(* IEC 61131-3 sources: repolevel_ST_code_completion/dataset/project_code/轴控/FB105_轴控制集/FC10_设备轴类, 3 files *)

(* ---- A01_通讯状态.st ---- *)
//从站通讯状态
pSlave := EtherCAT_Master_Leadshine.FirstSlave; //建立指针，指向主站后第一个从站
No_Slave:=0;
WHILE pSlave <> 0 DO
  No_Slave:=No_Slave+1;
  pSlave^(); //获取当前从站状态内容
IF pSlave^.wState <>ETC_SLAVE_STATE.ETC_SLAVE_OPERATIONAL THEN //
    ERROR[No_Slave]:=1;   //对应关系 ERROR[1]=1有错误   ERROR[1] 1号从站、ERROR[2] 2号从站,建立的数组元素个数等于从站个数
ELSE
    ERROR[No_Slave]:=0;
END_IF
pSlave := pSlave^.NextInstance; //指向下个从站，结尾为空，跳出循环
END_WHILE

//EtherCAT主站复位
EtherCAT_Master_Leadshine(
	xRestart:= bEtcReset,
	xStopBus:= ,
	xConfigFinished=> ,
	xDistributedClockInSync=> ,
	xError=> ,
	xSyncInWindow=> );

IF EtherCAT_Master_Leadshine.xConfigFinished AND EtherCAT_Master_Leadshine.xDistributedClockInSync THEN
	FB_AxisControl_AxisVirtual.ReStartSlaveEx:=TRUE;
	FB_AxisControl_调模A轴.ReStartSlaveEx:=TRUE;
	FB_AxisControl_调模B轴.ReStartSlaveEx:=TRUE;
	FB_AxisControl_送面料轴.ReStartSlaveEx:=TRUE;
	FB_AxisControl_取面料轴.ReStartSlaveEx:=TRUE;
	FB_AxisControl_横移A轴.ReStartSlaveEx:=TRUE;
	FB_AxisControl_升降A轴.ReStartSlaveEx:=TRUE;
	FB_AxisControl_横移B轴.ReStartSlaveEx:=TRUE;
	FB_AxisControl_升降B轴.ReStartSlaveEx:=TRUE;
	FB_AxisControl_出盒轴.ReStartSlaveEx:=TRUE;
	FB_AxisControl_铲灰板轴.ReStartSlaveEx:=TRUE;
	FB_AxisControl_包面纸轴.ReStartSlaveEx:=TRUE;
	FB_AxisControl_上包底轴.ReStartSlaveEx:=TRUE;
	FB_AxisControl_折边轴.ReStartSlaveEx:=TRUE;
	IF FB_AxisControl_AxisVirtual.ReStartSlaveDone AND FB_AxisControl_调模A轴.ReStartSlaveDone AND FB_AxisControl_调模B轴.ReStartSlaveDone AND
        FB_AxisControl_送面料轴.ReStartSlaveDone AND FB_AxisControl_取面料轴.ReStartSlaveDone AND FB_AxisControl_横移A轴.ReStartSlaveDone AND
		 FB_AxisControl_升降A轴.ReStartSlaveDone AND FB_AxisControl_横移B轴.ReStartSlaveDone AND FB_AxisControl_升降B轴.ReStartSlaveDone AND
		  FB_AxisControl_出盒轴.ReStartSlaveDone AND FB_AxisControl_铲灰板轴.ReStartSlaveDone AND FB_AxisControl_包面纸轴.ReStartSlaveDone AND
		   FB_AxisControl_上包底轴.ReStartSlaveDone AND FB_AxisControl_折边轴.ReStartSlaveDone THEN
	      bEtcReset:=FALSE;
	END_IF
END_IF

(* ---- A02_各轴状态.st ---- *)
(*EthercatBUS Cheak*)
IF b调模A轴通讯OK AND b调模B轴通讯OK AND b送面料轴通讯OK AND b取面料轴通讯OK AND b横移A轴通讯OK AND b升降A轴通讯OK AND
    b横移B轴通讯OK AND b升降B轴通讯OK AND b出盒轴通讯OK AND b铲灰板轴通讯OK AND b包面纸轴通讯OK AND b上包底轴通讯OK AND b折边轴通讯OK THEN
	b所有伺服总线通讯OK:=TRUE;
	ELSE
	b所有伺服总线通讯OK:=FALSE;
END_IF

IF b调模A轴使能OK AND b调模B轴使能OK AND b送面料轴使能OK AND b取面料轴使能OK AND b横移A轴使能OK AND b升降A轴使能OK AND
    b横移B轴使能OK AND b升降B轴使能OK AND b出盒轴使能OK AND b铲灰板轴使能OK AND b包面纸轴使能OK AND b上包底轴使能OK AND b折边轴使能OK THEN
	b所有伺服使能OK:=TRUE;
	ELSE
	b所有伺服使能OK:=FALSE;
END_IF

IF b调模A轴回零完成 AND b调模B轴回零完成 AND b送面料轴回零完成 AND b取面料轴回零完成 AND b横移A轴回零完成 AND b升降A轴回零完成 AND
    b横移B轴回零完成 AND b升降B轴回零完成 AND b出盒轴回零完成 AND b铲灰板轴回零完成 AND b包面纸轴回零完成 AND b上包底轴回零完成 AND b折边轴回零完成 THEN
	b所有伺服回零OK:=TRUE;
	ELSE
	b所有伺服回零OK:=FALSE;
END_IF

IF b调模A轴停止中 AND b调模B轴停止中 AND b送面料轴停止中 AND b取面料轴停止中 AND b横移A轴停止中 AND b升降A轴停止中 AND
    b横移B轴停止中 AND b升降B轴停止中 AND b出盒轴停止中 AND b铲灰板轴停止中 AND b包面纸轴停止中 AND b上包底轴停止中 AND b折边轴停止中 THEN
	b所有伺服静止中:=TRUE;
	ELSE
	b所有伺服静止中:=FALSE;
END_IF

(* ---- FC10_设备轴类.st ---- *)
PROGRAM FC10_设备轴类
VAR
	pSlave: POINTER TO ETCSlave;
    No_Slave: INT;
	bEtcReset: BOOL;

END_VAR

VAR_OUTPUT
	ERROR: ARRAY[1..13] OF INT;
END_VAR

A01_通讯状态();
A02_各轴状态();

FB50_虚轴控制();
FB51_调模A轴控制();
FB52_调模B轴控制();
FB53_送面料轴控制();
FB54_取面料轴控制();
FB55_横移A轴控制();
FB56_升降A轴控制();
FB57_横移B轴控制();
FB58_升降B轴控制();
FB59_出盒轴控制();
FB60_铲灰板轴控制();
FB61_包面纸轴控制();
FB62_上包底轴控制();
FB63_折边轴控制();
